FUNCTION_BLOCK EV_NeedleAxis (* Typed view of NeedleAxis's state channel (inputs and holder) *)
  (* Standard: 61499-2 *)
  (* Version 0.1, 2026-09-28, Project contributors, AAU Smart Production Lab *)
  PACKAGE filling;
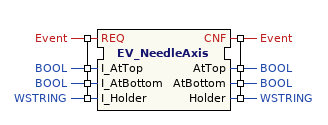
  EVENT_INPUT
    REQ WITH I_AtTop, I_AtBottom, I_Holder;
  END_EVENT
  EVENT_OUTPUT
    CNF WITH AtTop, AtBottom, Holder;
  END_EVENT
  VAR_INPUT
    I_AtTop : BOOL;
    I_AtBottom : BOOL;
    I_Holder : WSTRING;
  END_VAR
  VAR_OUTPUT
    AtTop : BOOL;
    AtBottom : BOOL;
    Holder : WSTRING;
  END_VAR
  EC_STATES
    REQ : REQ -> CNF;
  END_STATES
  ALGORITHM REQ IN ST:
AtTop := I_AtTop;
AtBottom := I_AtBottom;
Holder := I_Holder;
  END_ALGORITHM
END_FUNCTION_BLOCK
